(* CODESYS project LD_BASIC_OPTS.project

Project tree, tasks and I/O mapping:
  Device : AC702, Shenzhen Inovance Technology Co., Ltd., version 3.5.11.51
    application Application
      libraries: Standard, * (System)
      task MainTask (cyclic, interval 2000 ms, priority 2) calls PLC_PRG
      program PLC_PRG [LD]
      DifferentialMonitor
    HardWare Configuration
    Network Configuration
    Device Diagnosis
    Resources List
    ConfigStorage
    SoftMotion General Axis Pool
    LocalHSIO : 本地高速IO, 汇川技术股份有限公司, version 1.0.0.0
        unmapped channels: DigitalInput, DigitalOutput
    MODBUS_TCP : ModbusTCP本地从站, inovance, version 00.00.00.10
    HwConfiguratioinDevice : SystemConfig, Inovance, version 00.00.00.10
        settings: NetworkConfigArray.NetworkConfigArray.BusType = 10; NetworkConfigArray.NetworkConfigArray.RackSum = 1; NetworkConfigArray.NetworkConfigArray.HardwareConfigArray.HardwareConfigArray.RackNo = 1
*)

// Device/Application/PLC_PRG
PROGRAM PLC_PRG
VAR
	con1: BOOL := TRUE;
	out1: INT;
	res: INT;
	R_TRIG0: R_TRIG;
	TON0: TON;
	con2: BOOL;
END_VAR
VAR // added by the converter: edge detectors and wires of the graphical bodies
    _w1, _w2 : BOOL;
END_VAR

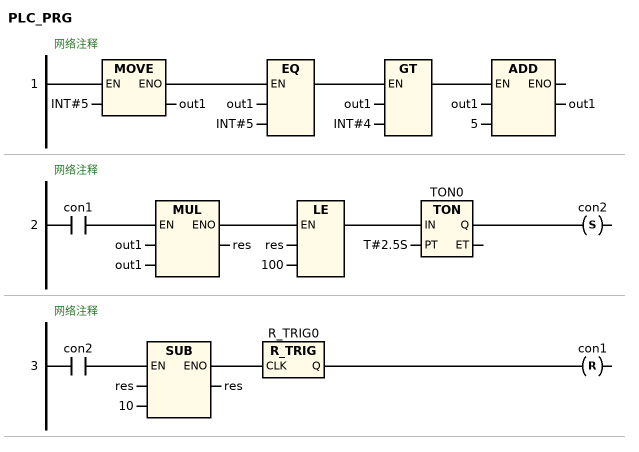
// NETWORK 1
// 网络注释
out1 := INT#5;
IF out1 = INT#5 AND out1 > INT#4 THEN out1 := out1 + 5; END_IF

// NETWORK 2
// 网络注释
_w1 := con1;
IF _w1 THEN res := out1 * out1; END_IF
TON0(IN := _w1 AND res <= 100, PT := T#2.5S); // TON
con2 S= TON0.Q;

// NETWORK 3
// 网络注释
_w2 := con2;
IF _w2 THEN res := res - 10; END_IF
R_TRIG0(CLK := _w2); // R_TRIG
con1 R= R_TRIG0.Q;

END_PROGRAM
